FUNCTION_BLOCK ATURNTABLE_DEMUX (* Composite FB wrapping other FBs *)
  (* Standard: 61499-2 *)
  (* Version 0.0, 2008-07-10, 4DIAC-IDE, 4DIAC-Consortium *)
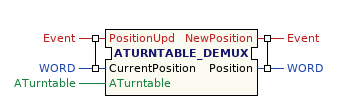
  EVENT_INPUT
    PositionUpd WITH CurrentPosition; (* Request from Socket *)
  END_EVENT
  EVENT_OUTPUT
    NewPosition WITH Position; (* Confirmation from Plug *)
  END_EVENT
  VAR_INPUT
    CurrentPosition : WORD; (* Request Data from Socket *)
  END_VAR
  VAR_OUTPUT
    Position : WORD; (* Confirmation Data from Plug *)
  END_VAR
  SOCKETS
    ATurntable : ATurntable;
  END_SOCKETS
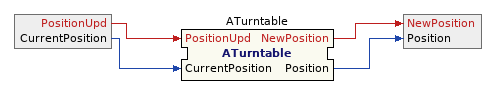
  EVENT_CONNECTIONS
    PositionUpd TO ATurntable.PositionUpd;
    ATurntable.NewPosition TO NewPosition;
  END_CONNECTIONS
  DATA_CONNECTIONS
    CurrentPosition TO ATurntable.CurrentPosition;
    ATurntable.Position TO Position;
  END_CONNECTIONS
END_FUNCTION_BLOCK
